KUKA KRL program: HandGuiding_TargetTeaching.src, HandGuiding_TargetTeaching.dat

--- HandGuiding_TargetTeaching.src ---
&ACCESS RVO
&REL 1
&PARAM DISKPATH = KRC:\R1\Program\ForceTorqueSensor
DEF HandGuide_record_pt ( )
   DECL INT counter


   GLOBAL INTERRUPT DECL 3 WHEN $STOPMESS==TRUE DO IR_STOPM ( )
   INTERRUPT ON 3
   BAS (#INITMOV,0 )

   PTP $AXIS_ACT

   ; Base in actual position
   $BASE.X=$POS_ACT.X
   $BASE.Y=$POS_ACT.Y
   $BASE.Z=$POS_ACT.Z
   $BASE.A=$POS_ACT.A
   $BASE.B=$POS_ACT.B
   $BASE.C=$POS_ACT.C

   ; 0 Values Initialization
   $SEN_PREA[1]=-myF0[1]
   $SEN_PREA[2]=-myF0[2]
   $SEN_PREA[3]=-myF0[3]
   $SEN_PREA[4]=-myM0[1]
   $SEN_PREA[5]=-myM0[2]
   $SEN_PREA[6]=-myM0[3]
   $SEN_PREA[7]=TOOL_WEIGHT
   $SEN_PREA[8]=POS_CG[1]
   $SEN_PREA[9]=POS_CG[2]
   $SEN_PREA[10]=POS_CG[3]

   ; Sensor guided movement
   counter = 0
   REPEAT
      counter = counter + 1
      StartHG()
      WAIT FOR $IN[4]
      myPos[counter].X = $POS_ACT.X
      myPos[counter].Y = $POS_ACT.Y
      myPos[counter].Z = $POS_ACT.Z
      myPos[counter].A = $POS_ACT.A
      myPos[counter].B = $POS_ACT.B
      myPos[counter].C = $POS_ACT.C
      myPos[counter].S = $POS_ACT.S
      myPos[counter].T = $POS_ACT.T

      ; Or via SEN_PREA if taken from RSI block (POS_ACT)

      WAIT FOR NOT($IN[4])
   UNTIL (counter == n_measures )

   ; Move back to start position
   PTP {A1 0, A2 -130, A3 130, A4 0, A5 90, A6 0}

END



DEF StartHG()

   DECL INT ret	; Return value for RSI commands
   DECL INT CONTID	; ContainerID

   ret=RSI_CREATE("HandGuiding_record_pt.rsi",CONTID)
   IF (ret <> RSIOK) THEN
      HALT
   ENDIF

   ; Start RSI execution
   ret=RSI_ON(#RELATIVE,#IPO_FAST)
   IF (ret <> RSIOK) THEN
      HALT
   ENDIF

   RSI_MOVECORR()

   ; Turn off RSI
   ret=RSI_OFF()
   IF (ret <> RSIOK) THEN
      HALT
   ENDIF
END

--- HandGuiding_TargetTeaching.dat ---
&ACCESS RVO
DEFDAT  HandGuide_record_pt PUBLIC
; Settings
DECL INT n_measures=10
DECL POS myPos[10]

; Data
myPos[1]={X 6.39245033,Y -460.911133,Z -13.2861853,A 2.48526049,B -2.33426857,C -0.999733686,S 18,T 11}
myPos[2]={X 37.2615929,Y -553.389160,Z 457.148346,A 1.72387600,B -1.16733873,C 0.449589849,S 18,T 3}
myPos[3]={X 0.0,Y 0.0,Z 0.0,A 0.0,B 0.0,C 0.0,S 0,T 0}
myPos[4]={X 0.0,Y 0.0,Z 0.0,A 0.0,B 0.0,C 0.0,S 0,T 0}
myPos[5]={X 0.0,Y 0.0,Z 0.0,A 0.0,B 0.0,C 0.0,S 0,T 0}
myPos[6]={X 0.0,Y 0.0,Z 0.0,A 0.0,B 0.0,C 0.0,S 0,T 0}
myPos[7]={X 0.0,Y 0.0,Z 0.0,A 0.0,B 0.0,C 0.0,S 0,T 0}
myPos[8]={X 0.0,Y 0.0,Z 0.0,A 0.0,B 0.0,C 0.0,S 0,T 0}
myPos[9]={X 0.0,Y 0.0,Z 0.0,A 0.0,B 0.0,C 0.0,S 0,T 0}
myPos[10]={X 0.0,Y 0.0,Z 0.0,A 0.0,B 0.0,C 0.0,S 0,T 0}
ENDDAT
